// Mitsubishi GX Works2 project: PLC_GROUP12   PLC: FX3G

// global labels: Global1
VAR_GLOBAL
  startDay AT X007 : BOOL;
  WorkingDay AT Y007 : BOOL;
  EmergencySwitch AT X005 : BOOL;
  IceCreamMake AT X001 : BOOL;
END_VAR
VAR_GLOBAL CONSTANT
  Div_Mul_400 : REAL := 400;
END_VAR
VAR_GLOBAL
  regularIceLight AT M10 : BOOL;
END_VAR
VAR_GLOBAL CONSTANT
  MaxForRegular_5 : REAL := 5;
END_VAR
VAR_GLOBAL
  typeInput AT D1300 : REAL;
  analog_Input1 AT D8280 : INT;
  pinukIceLight AT M11 : BOOL;
  PetelAmount AT D1400 : REAL;
  LimonAmount AT D1410 : REAL;
  StableAmount AT D1420 : REAL;
  GummyAmount AT D1430 : REAL;
END_VAR
VAR_GLOBAL CONSTANT
  BearsForRegular_28 : REAL := 28;
END_VAR
VAR_GLOBAL
  EnoughForRegular AT M5 : BOOL;
END_VAR
VAR_GLOBAL CONSTANT
  BearsForPinuk_70 : REAL := 70;
END_VAR
VAR_GLOBAL
  EnoughForPinuk AT M6 : BOOL;
  PetelIcecream AT D1500 : REAL;
END_VAR
VAR_GLOBAL CONSTANT
  PetelIcecream_R_350 : REAL := 350;
  LemonIcecream_R_490 : REAL := 490;
END_VAR
VAR_GLOBAL
  LemonIcecream AT D1510 : REAL;
  StartMakingRegular AT M21 : BOOL;
END_VAR
VAR_GLOBAL CONSTANT
  PetelIcecream_P_560 : REAL := 560;
  LemonIcecream_P_700 : REAL := 700;
  LemonForRegular_455 : REAL := 455;
  StableForRegular_105 : REAL := 105;
END_VAR
VAR_GLOBAL
  subInvRegular AT M7 : BOOL;
  subInvPinuk AT M8 : BOOL;
END_VAR
VAR_GLOBAL CONSTANT
  PetelForPinuk_385 : REAL := 385;
  LemonForPinuk_665 : REAL := 665;
  StableForPinuk_210 : REAL := 210;
  IceCreamTimer_50 : INT := 50;
END_VAR
VAR_GLOBAL
  TimerForIceCream AT TC1 : BOOL;
  FinishedIceCream AT TS1 : BOOL;
  IceCreamMakeLight AT Y000 : BOOL;
  StartMakingPinuk AT M22 : BOOL;
  startFridge AT X002 : BOOL;
  PetelFridge AT D1600 : REAL;
  LemonFridge AT D1610 : REAL;
  MoveToFridge AT M23 : BOOL;
END_VAR
VAR_GLOBAL CONSTANT
  FridgeTimer_80 : INT := 80;
END_VAR
VAR_GLOBAL
  TimerForFridge AT TC2 : BOOL;
  FinishedFridge AT TS2 : BOOL;
  tempSensor AT X003 : BOOL;
  IceCreamFridgeLight AT Y002 : BOOL;
END_VAR
VAR_GLOBAL CONSTANT
  MinForPinuk_6 : REAL := 6;
END_VAR
VAR_GLOBAL
  EnoughInventoryPinuk AT M9 : BOOL;
  EnoughInventoryRegular AT M4 : BOOL;
  mixConatainer AT D1666 : REAL;
  BlendRegular AT M30 : BOOL;
  BlendPinuk AT M31 : BOOL;
  StartBlink AT M32 : BOOL;
END_VAR
VAR_GLOBAL CONSTANT
  SingleBlink_3 : INT := 3;
END_VAR
VAR_GLOBAL
  TimerForOneBlinkY5 AT TC3 : BOOL;
  FinishedOneBlinkY5 AT TS3 : BOOL;
  MixLight1 AT Y005 : BOOL;
  TimerForOneBlinkY6 AT TC4 : BOOL;
  FinishedOneBlinkY6 AT TS4 : BOOL;
  MixLight2 AT Y006 : BOOL;
  FinishedBlendReg AT TS5 : BOOL;
  TimerForBlendReg AT TC5 : BOOL;
END_VAR
VAR_GLOBAL CONSTANT
  BlinkRegular_30 : INT := 30;
END_VAR
VAR_GLOBAL
  BlinkRegular AT M45 : BOOL;
  BlinkPinuk AT M46 : BOOL;
  FinishedBlendPinuk AT TS6 : BOOL;
END_VAR
VAR_GLOBAL CONSTANT
  BlinkPinuk_50 : INT := 50;
END_VAR
VAR_GLOBAL
  TimerForBlendPinuk AT TC6 : BOOL;
  StartPacking AT X004 : BOOL;
  GummyPack AT X000 : BOOL;
  CounterForPacking AT CC1 : BOOL;
END_VAR
VAR_GLOBAL CONSTANT
  UnitsCounter_7 : INT := 7;
END_VAR
VAR_GLOBAL
  FinishedPacking AT CS1 : BOOL;
  PackUnit AT Y004 : BOOL;
  Storage AT D1700 : REAL;
END_VAR
VAR_GLOBAL CONSTANT
  ReadyPackage_1 : REAL := 1;
  OutputDivider_10 : REAL := 10;
END_VAR
VAR_GLOBAL
  output AT D1710 : REAL;
  analogOutput AT D8282 : INT;
END_VAR
VAR_GLOBAL CONSTANT
  RegularUnit_124 : REAL := 124;
  PinukUnit_190 : REAL := 190;
  PetelForRegular_280 : REAL := 280;
END_VAR
VAR_GLOBAL
  EndIteration AT M59 : BOOL;
  NoInventory AT M60 : BOOL;
  RegistorZero AT D1800 : REAL;
  RegZero AT D1810 : INT;
END_VAR
VAR_GLOBAL CONSTANT
  PetelForRegular_279 : REAL := 279;
  LemonForRegular_454 : REAL := 454;
  StableForRegular_104 : REAL := 104;
  BearsForRegular_27 : REAL := 27;
END_VAR

// task Task_01 (event TRUE, interval 0, priority 31): POU_01

PROGRAM POU_01
(* structured ladder/FBD written out as ST: instructions are called as NAME(EN, inputs, outputs); _pN, _eN, _tN stand for wires *)
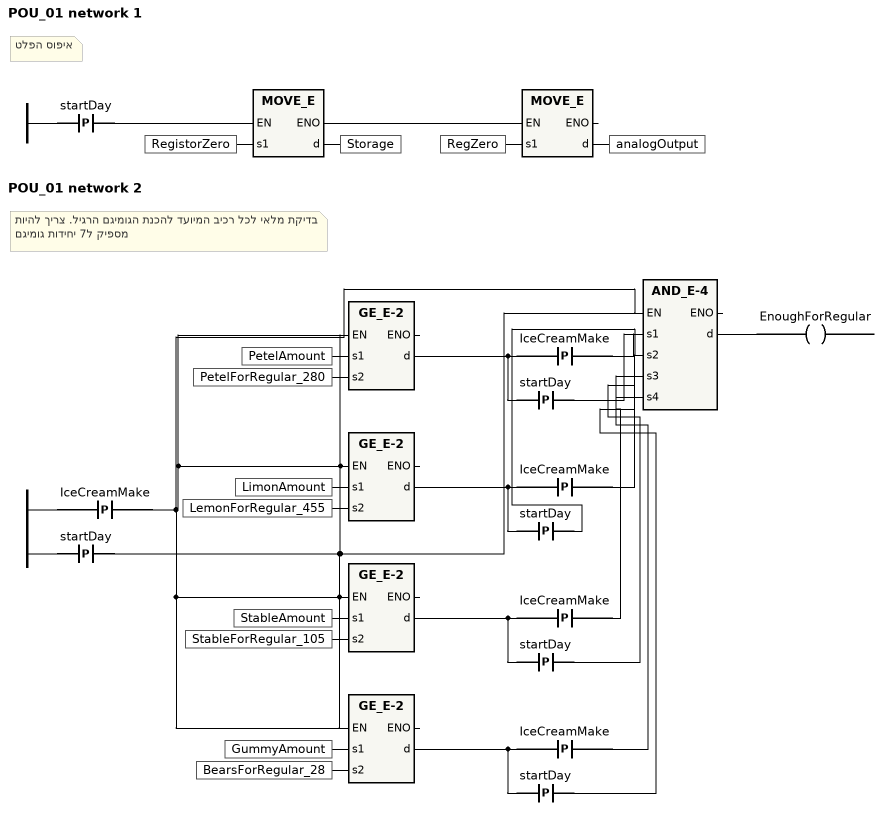
(* network 1 *)
(* איפוס הפלט *)
_e1 := MOVE_E(LDP(TRUE, startDay), RegistorZero, Storage);
MOVE_E(_e1, RegZero, analogOutput);
(* network 2 *)
(* בדיקת מלאי לכל רכיב המיועד להכנת הגומיגם הרגיל. צריך להיות מספיק ל7 יחידות גומיגם *)
_p1 := LDP(TRUE, IceCreamMake) OR LDP(TRUE, startDay);
GE_E(_p1, PetelAmount, PetelForRegular_280, _t2);
GE_E(_p1, LimonAmount, LemonForRegular_455, _t3);
GE_E(_p1, StableAmount, StableForRegular_105, _t4);
GE_E(_p1, GummyAmount, BearsForRegular_28, _t5);
AND_E(_p1, (_t2 AND LDP(TRUE, IceCreamMake)) OR (_t2 AND LDP(TRUE, startDay)), (_t3 AND LDP(TRUE, IceCreamMake)) OR (_t3 AND LDP(TRUE, startDay)), (_t4 AND LDP(TRUE, IceCreamMake)) OR (_t4 AND LDP(TRUE, startDay)), (_t5 AND LDP(TRUE, IceCreamMake)) OR (_t5 AND LDP(TRUE, startDay)), _t6);
EnoughForRegular := _t6;
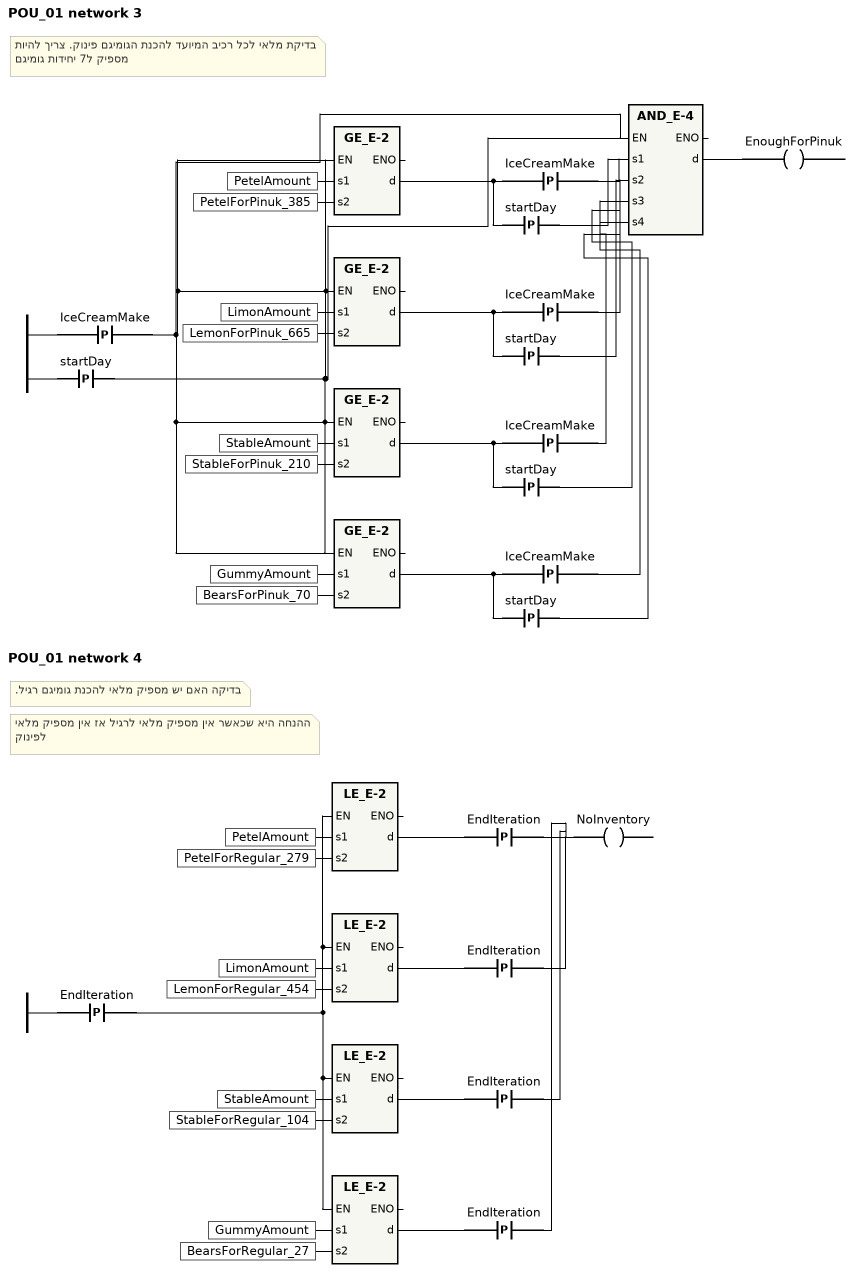
(* network 3 *)
(* בדיקת מלאי לכל רכיב המיועד להכנת הגומיגם פינוק. צריך להיות מספיק ל7 יחידות גומיגם *)
_p1 := LDP(TRUE, IceCreamMake) OR LDP(TRUE, startDay);
GE_E(_p1, PetelAmount, PetelForPinuk_385, _t2);
GE_E(_p1, LimonAmount, LemonForPinuk_665, _t3);
GE_E(_p1, StableAmount, StableForPinuk_210, _t4);
GE_E(_p1, GummyAmount, BearsForPinuk_70, _t5);
AND_E(_p1, (_t2 AND LDP(TRUE, IceCreamMake)) OR (_t2 AND LDP(TRUE, startDay)), (_t3 AND LDP(TRUE, IceCreamMake)) OR (_t3 AND LDP(TRUE, startDay)), (_t4 AND LDP(TRUE, IceCreamMake)) OR (_t4 AND LDP(TRUE, startDay)), (_t5 AND LDP(TRUE, IceCreamMake)) OR (_t5 AND LDP(TRUE, startDay)), _t6);
EnoughForPinuk := _t6;
(* network 4 *)
(* בדיקה האם יש מספיק מלאי להכנת גומיגם רגיל. *)
(* ההנחה היא שכאשר אין מספיק מלאי לרגיל אז אין מספיק מלאי לפינוק *)
_p1 := LDP(TRUE, EndIteration);
LE_E(_p1, PetelAmount, PetelForRegular_279, _t2);
LE_E(_p1, LimonAmount, LemonForRegular_454, _t3);
LE_E(_p1, StableAmount, StableForRegular_104, _t4);
LE_E(_p1, GummyAmount, BearsForRegular_27, _t5);
NoInventory := (_t2 AND LDP(TRUE, EndIteration)) OR (_t3 AND LDP(TRUE, EndIteration)) OR (_t4 AND LDP(TRUE, EndIteration)) OR (_t5 AND LDP(TRUE, EndIteration));
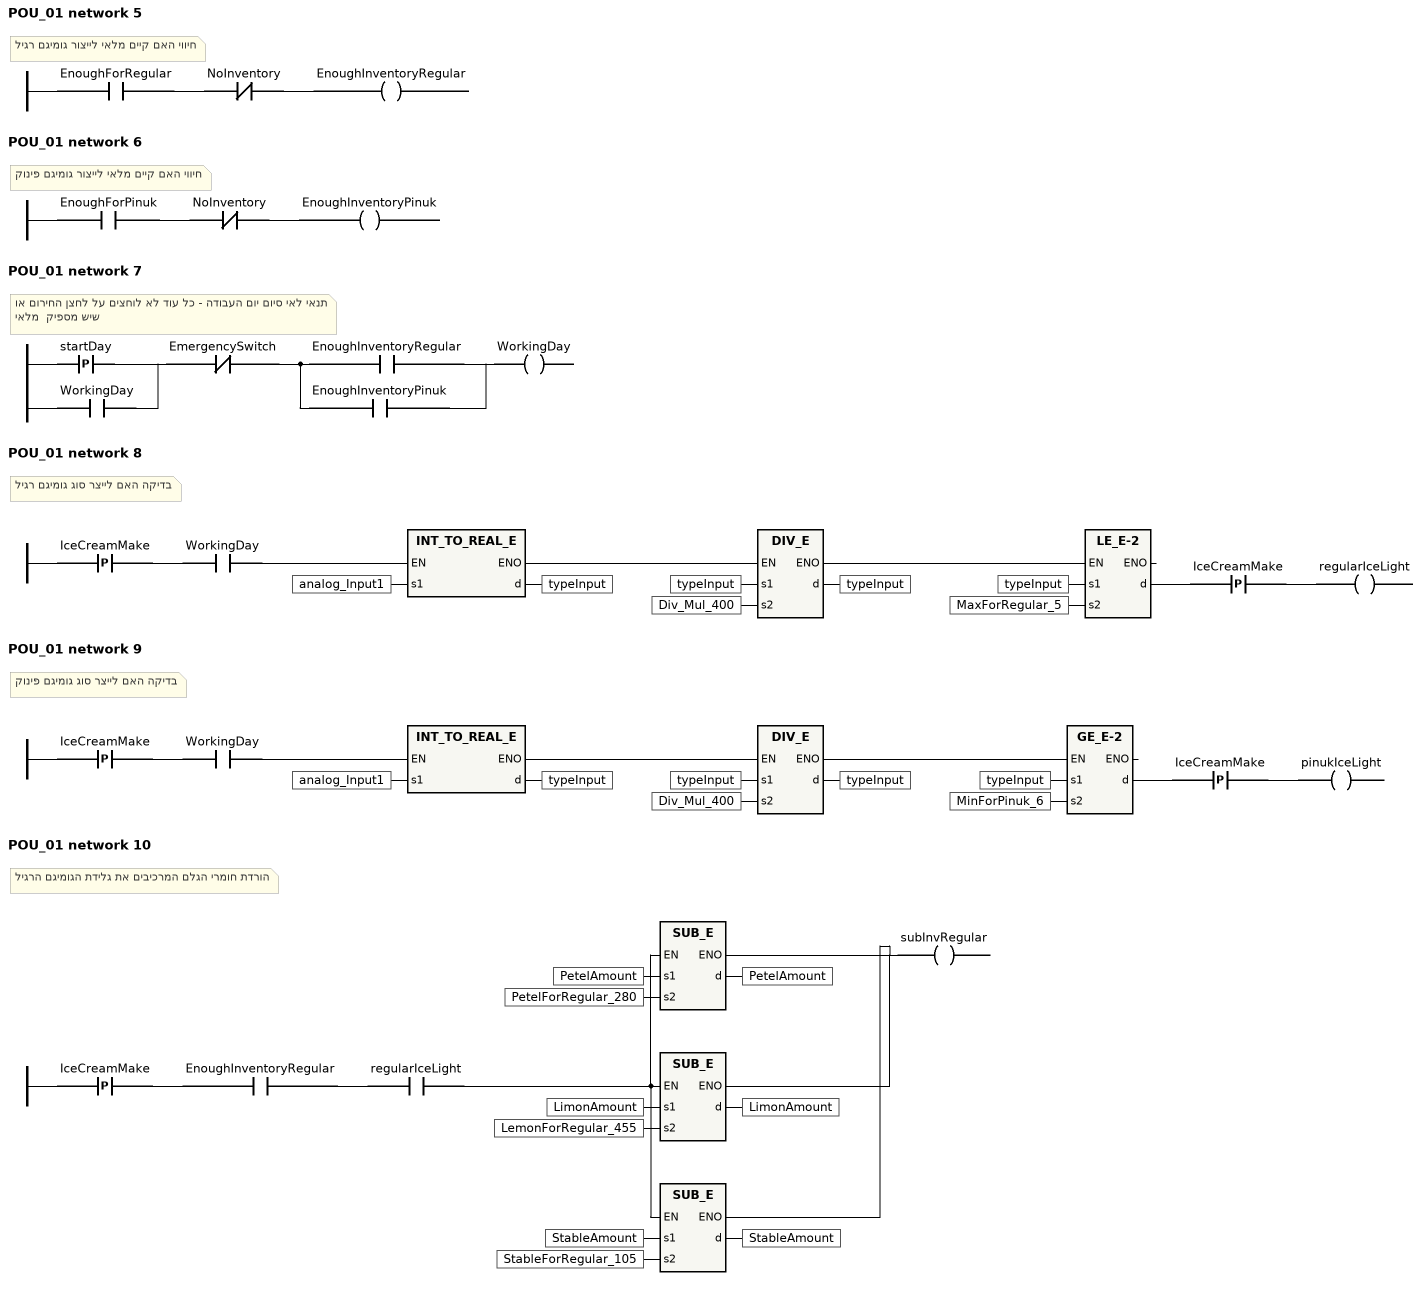
(* network 5 *)
(* חיווי האם קיים מלאי לייצור גומיגם רגיל *)
EnoughInventoryRegular := EnoughForRegular AND NOT NoInventory;
(* network 6 *)
(* חיווי האם קיים מלאי לייצור גומיגם פינוק *)
EnoughInventoryPinuk := EnoughForPinuk AND NOT NoInventory;
(* network 7 *)
(* תנאי לאי סיום יום העבודה - כל עוד לא לוחצים על לחצן החירום או שיש מספיק  מלאי *)
_p1 := (LDP(TRUE, startDay) OR WorkingDay) AND NOT EmergencySwitch;
WorkingDay := (_p1 AND EnoughInventoryRegular) OR (_p1 AND EnoughInventoryPinuk);
(* network 8 *)
(* בדיקה האם לייצר סוג גומיגם רגיל *)
_e1 := INT_TO_REAL_E(LDP(TRUE, IceCreamMake) AND WorkingDay, analog_Input1, typeInput);
_e2 := DIV_E(_e1, typeInput, Div_Mul_400, typeInput);
LE_E(_e2, typeInput, MaxForRegular_5, _t3);
regularIceLight := _t3 AND LDP(TRUE, IceCreamMake);
(* network 9 *)
(* בדיקה האם לייצר סוג גומיגם פינוק *)
_e1 := INT_TO_REAL_E(LDP(TRUE, IceCreamMake) AND WorkingDay, analog_Input1, typeInput);
_e2 := DIV_E(_e1, typeInput, Div_Mul_400, typeInput);
GE_E(_e2, typeInput, MinForPinuk_6, _t3);
pinukIceLight := _t3 AND LDP(TRUE, IceCreamMake);
(* network 10 *)
(* הורדת חומרי הגלם המרכיבים את גלידת הגומיגם הרגיל *)
_p1 := LDP(TRUE, IceCreamMake) AND EnoughInventoryRegular AND regularIceLight;
_e2 := SUB_E(_p1, PetelAmount, PetelForRegular_280, PetelAmount);
_e3 := SUB_E(_p1, LimonAmount, LemonForRegular_455, LimonAmount);
_e4 := SUB_E(_p1, StableAmount, StableForRegular_105, StableAmount);
subInvRegular := _e2 OR _e3 OR _e4;
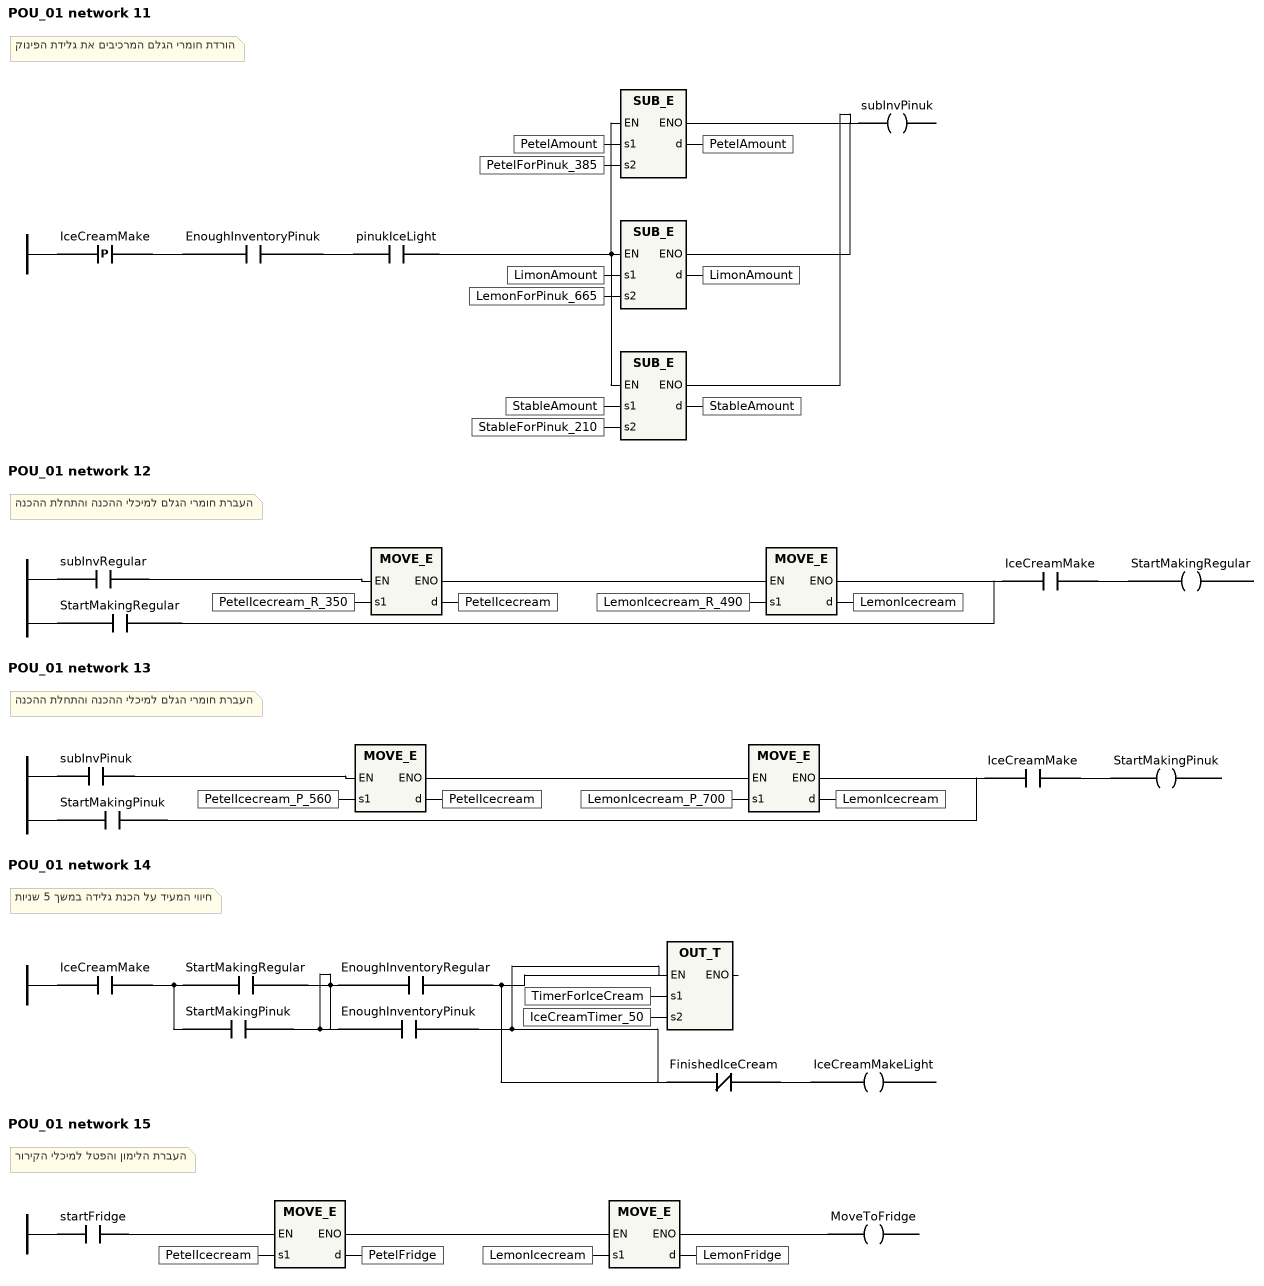
(* network 11 *)
(* הורדת חומרי הגלם המרכיבים את גלידת הפינוק *)
_p1 := LDP(TRUE, IceCreamMake) AND EnoughInventoryPinuk AND pinukIceLight;
_e2 := SUB_E(_p1, PetelAmount, PetelForPinuk_385, PetelAmount);
_e3 := SUB_E(_p1, LimonAmount, LemonForPinuk_665, LimonAmount);
_e4 := SUB_E(_p1, StableAmount, StableForPinuk_210, StableAmount);
subInvPinuk := _e2 OR _e3 OR _e4;
(* network 12 *)
(* העברת חומרי הגלם למיכלי ההכנה והתחלת ההכנה *)
_e1 := MOVE_E(subInvRegular, PetelIcecream_R_350, PetelIcecream);
_e2 := MOVE_E(_e1, LemonIcecream_R_490, LemonIcecream);
StartMakingRegular := (_e2 OR StartMakingRegular) AND IceCreamMake;
(* network 13 *)
(* העברת חומרי הגלם למיכלי ההכנה והתחלת ההכנה *)
_e1 := MOVE_E(subInvPinuk, PetelIcecream_P_560, PetelIcecream);
_e2 := MOVE_E(_e1, LemonIcecream_P_700, LemonIcecream);
StartMakingPinuk := (_e2 OR StartMakingPinuk) AND IceCreamMake;
(* network 14 *)
(* חיווי המעיד על הכנת גלידה במשך 5 שניות *)
_p1 := (IceCreamMake AND StartMakingRegular) OR (IceCreamMake AND StartMakingPinuk);
_p2 := (_p1 AND EnoughInventoryRegular) OR (_p1 AND EnoughInventoryPinuk);
IceCreamMakeLight := _p2 AND NOT FinishedIceCream;
OUT_T(_p2, TimerForIceCream, IceCreamTimer_50);
(* network 15 *)
(* העברת הלימון והפטל למיכלי הקירור *)
_e1 := MOVE_E(startFridge, PetelIcecream, PetelFridge);
_e2 := MOVE_E(_e1, LemonIcecream, LemonFridge);
MoveToFridge := _e2;
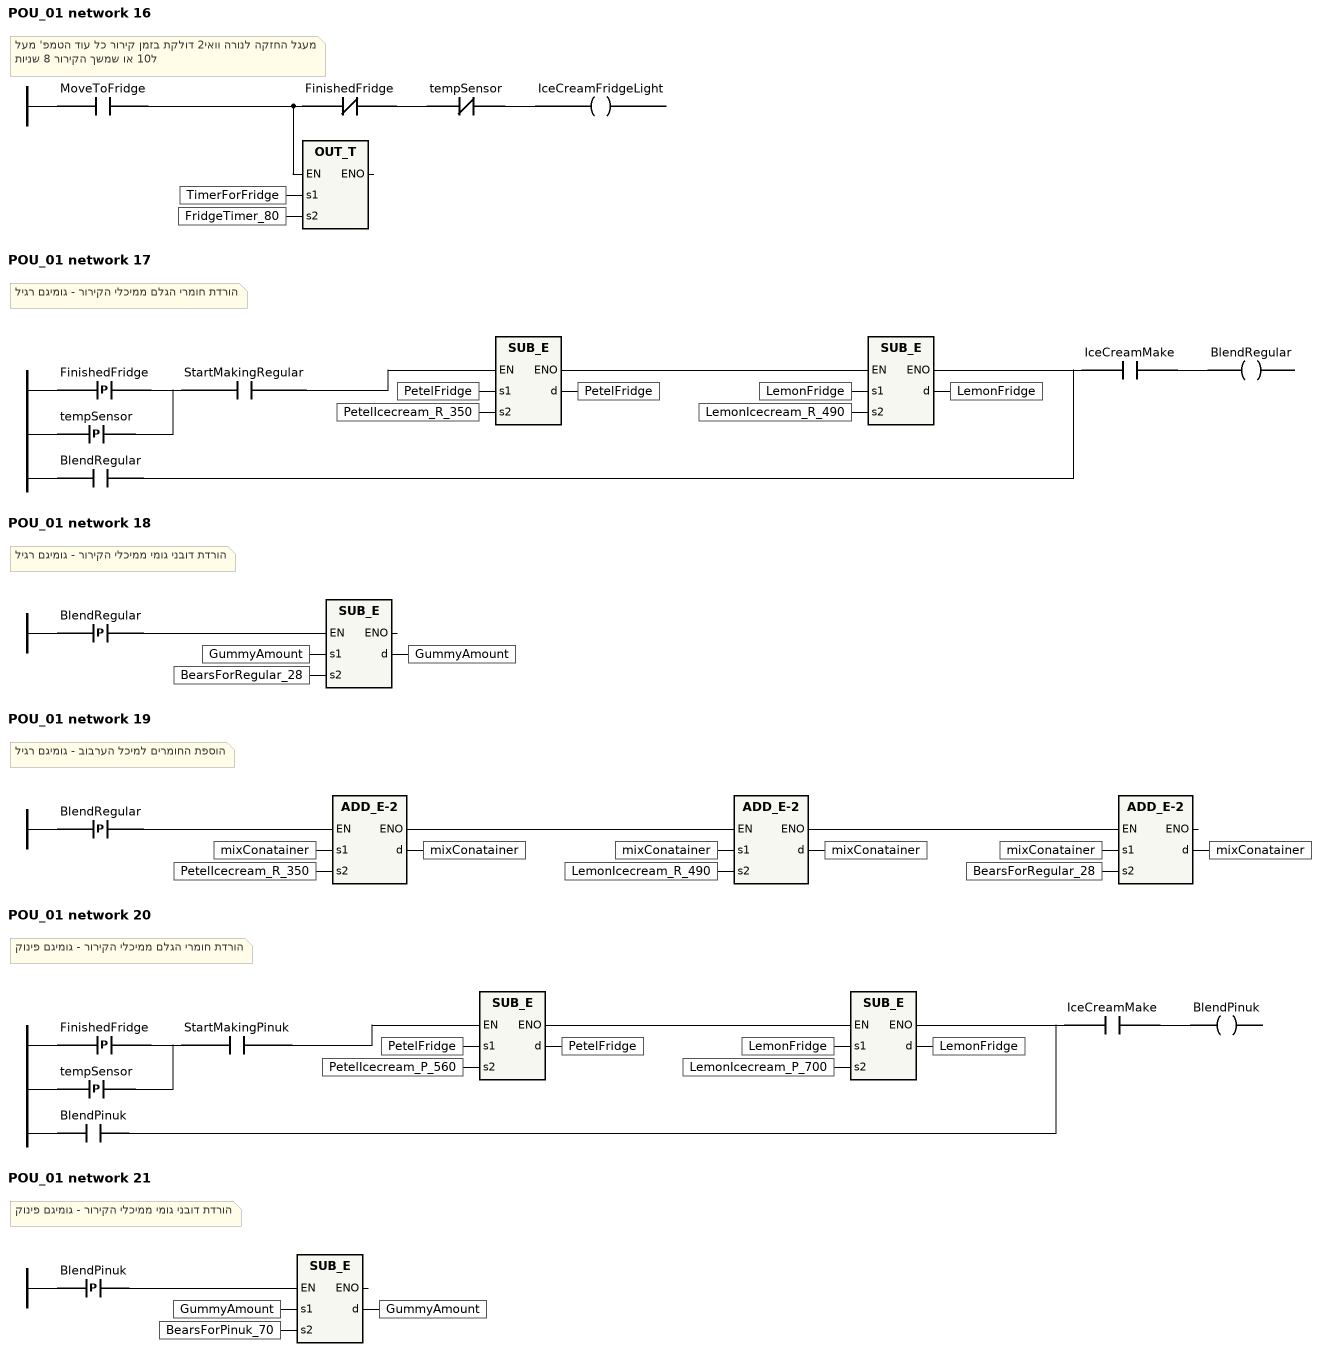
(* network 16 *)
(* מעגל החזקה לנורה וואי2 דולקת בזמן קירור כל עוד הטמפ' מעל ל10 או שמשך הקירור 8 שניות *)
IceCreamFridgeLight := MoveToFridge AND NOT FinishedFridge AND NOT tempSensor;
OUT_T(MoveToFridge, TimerForFridge, FridgeTimer_80);
(* network 17 *)
(* הורדת חומרי הגלם ממיכלי הקירור - גומיגם רגיל *)
_e1 := SUB_E((LDP(TRUE, FinishedFridge) OR LDP(TRUE, tempSensor)) AND StartMakingRegular, PetelFridge, PetelIcecream_R_350, PetelFridge);
_e2 := SUB_E(_e1, LemonFridge, LemonIcecream_R_490, LemonFridge);
BlendRegular := (_e2 OR BlendRegular) AND IceCreamMake;
(* network 18 *)
(* הורדת דובני גומי ממיכלי הקירור - גומיגם רגיל *)
SUB_E(LDP(TRUE, BlendRegular), GummyAmount, BearsForRegular_28, GummyAmount);
(* network 19 *)
(* הוספת החומרים למיכל הערבוב - גומיגם רגיל *)
_e1 := ADD_E(LDP(TRUE, BlendRegular), mixConatainer, PetelIcecream_R_350, mixConatainer);
_e2 := ADD_E(_e1, mixConatainer, LemonIcecream_R_490, mixConatainer);
ADD_E(_e2, mixConatainer, BearsForRegular_28, mixConatainer);
(* network 20 *)
(* הורדת חומרי הגלם ממיכלי הקירור - גומיגם פינוק *)
_e1 := SUB_E((LDP(TRUE, FinishedFridge) OR LDP(TRUE, tempSensor)) AND StartMakingPinuk, PetelFridge, PetelIcecream_P_560, PetelFridge);
_e2 := SUB_E(_e1, LemonFridge, LemonIcecream_P_700, LemonFridge);
BlendPinuk := (_e2 OR BlendPinuk) AND IceCreamMake;
(* network 21 *)
(* הורדת דובני גומי ממיכלי הקירור - גומיגם פינוק *)
SUB_E(LDP(TRUE, BlendPinuk), GummyAmount, BearsForPinuk_70, GummyAmount);
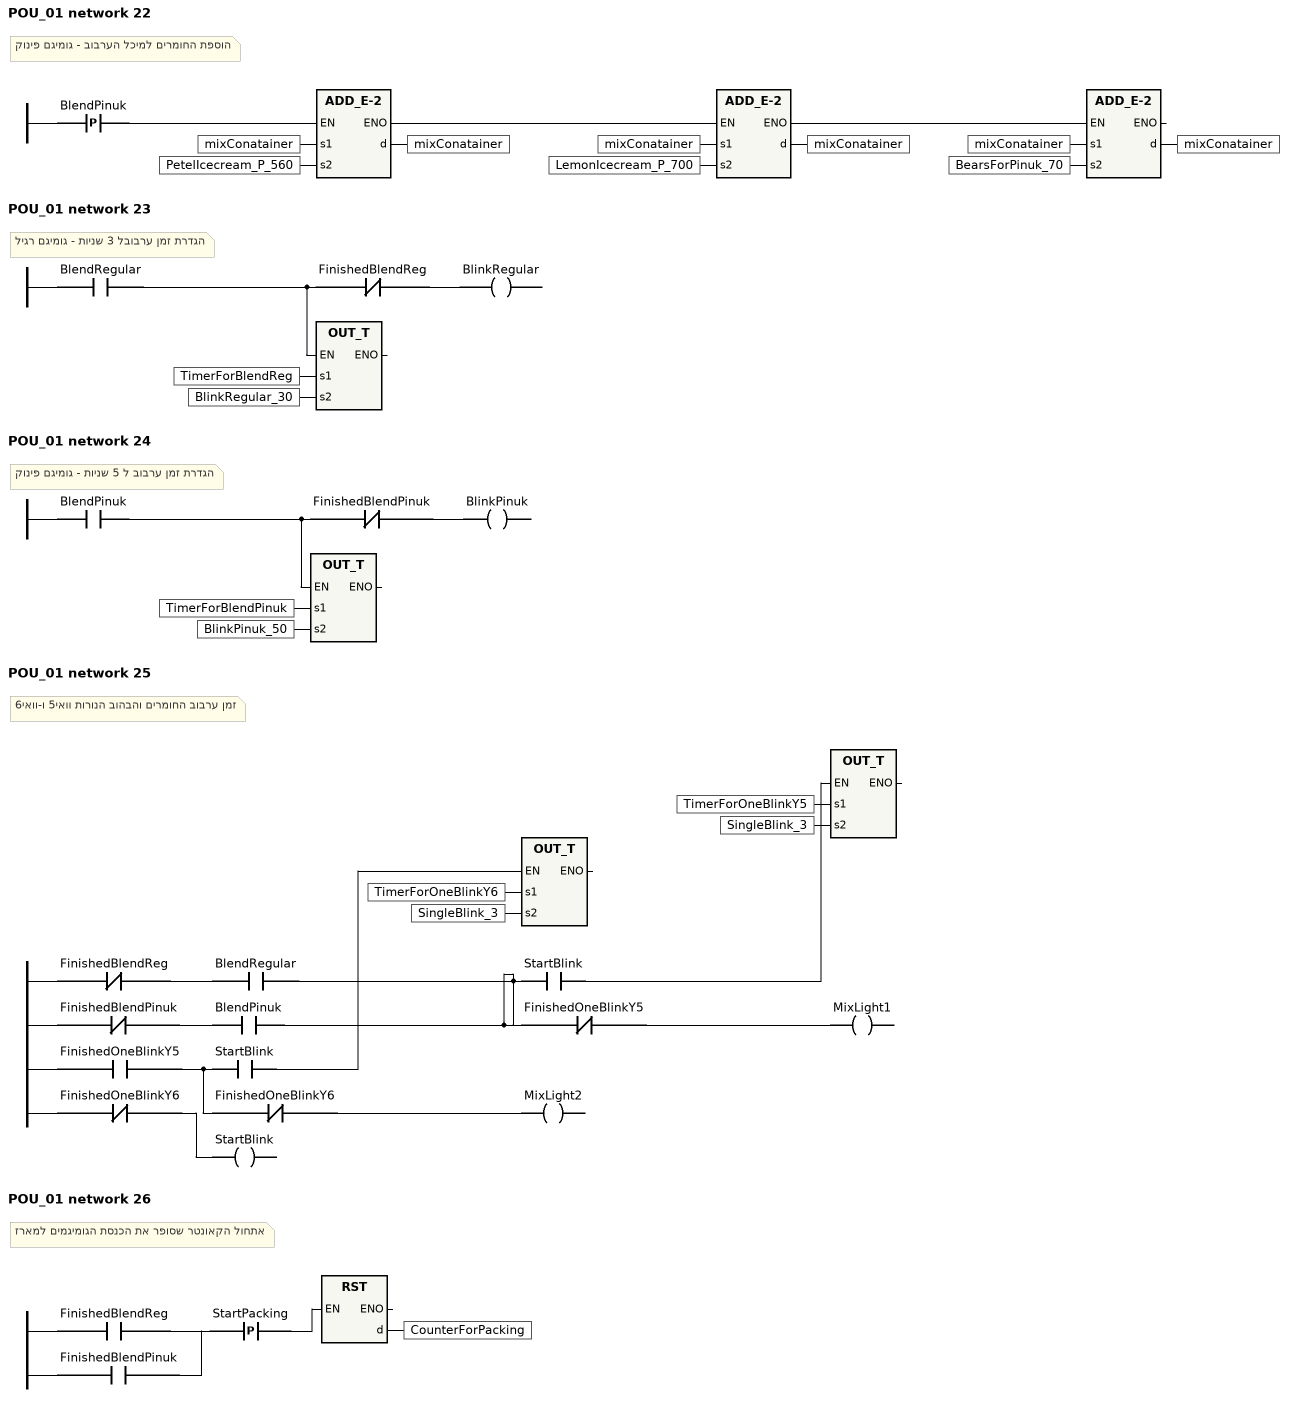
(* network 22 *)
(* הוספת החומרים למיכל הערבוב - גומיגם פינוק *)
_e1 := ADD_E(LDP(TRUE, BlendPinuk), mixConatainer, PetelIcecream_P_560, mixConatainer);
_e2 := ADD_E(_e1, mixConatainer, LemonIcecream_P_700, mixConatainer);
ADD_E(_e2, mixConatainer, BearsForPinuk_70, mixConatainer);
(* network 23 *)
(* הגדרת זמן ערבובל 3 שניות - גומיגם רגיל *)
BlinkRegular := BlendRegular AND NOT FinishedBlendReg;
OUT_T(BlendRegular, TimerForBlendReg, BlinkRegular_30);
(* network 24 *)
(* הגדרת זמן ערבוב ל 5 שניות - גומיגם פינוק *)
BlinkPinuk := BlendPinuk AND NOT FinishedBlendPinuk;
OUT_T(BlendPinuk, TimerForBlendPinuk, BlinkPinuk_50);
(* network 25 *)
(* זמן ערבוב החומרים והבהוב הנורות וואי5 ו-וואי6 *)
_p1 := (NOT FinishedBlendReg AND BlendRegular) OR (NOT FinishedBlendPinuk AND BlendPinuk);
OUT_T(_p1 AND StartBlink, TimerForOneBlinkY5, SingleBlink_3);
MixLight1 := _p1 AND NOT FinishedOneBlinkY5;
OUT_T(FinishedOneBlinkY5 AND StartBlink, TimerForOneBlinkY6, SingleBlink_3);
MixLight2 := FinishedOneBlinkY5 AND NOT FinishedOneBlinkY6;
StartBlink := NOT FinishedOneBlinkY6;
(* network 26 *)
(* אתחול הקאונטר שסופר את הכנסת הגומיגמים למארז *)
RST((FinishedBlendReg OR FinishedBlendPinuk) AND LDP(TRUE, StartPacking), CounterForPacking);
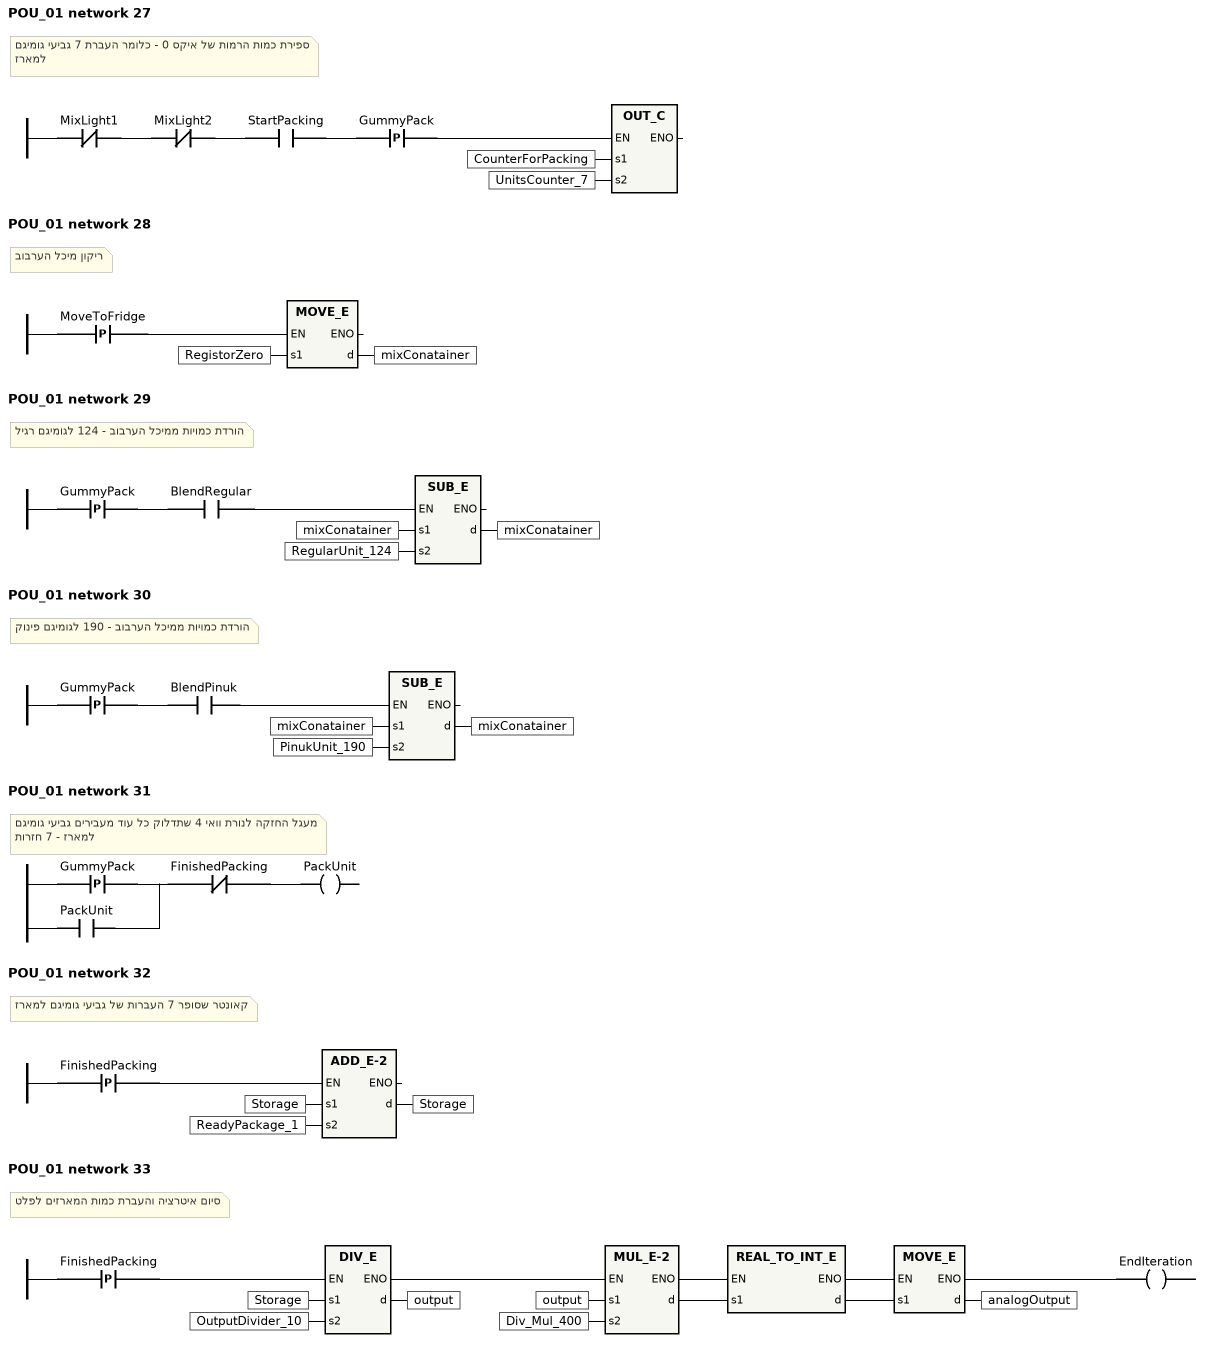
(* network 27 *)
(* ספירת כמות הרמות של איקס 0 - כלומר העברת 7 גביעי גומיגם למארז *)
OUT_C(NOT MixLight1 AND NOT MixLight2 AND StartPacking AND LDP(TRUE, GummyPack), CounterForPacking, UnitsCounter_7);
(* network 28 *)
(* ריקון מיכל הערבוב *)
MOVE_E(LDP(TRUE, MoveToFridge), RegistorZero, mixConatainer);
(* network 29 *)
(* הורדת כמויות ממיכל הערבוב - 124 לגומיגם רגיל *)
SUB_E(LDP(TRUE, GummyPack) AND BlendRegular, mixConatainer, RegularUnit_124, mixConatainer);
(* network 30 *)
(* הורדת כמויות ממיכל הערבוב - 190 לגומיגם פינוק *)
SUB_E(LDP(TRUE, GummyPack) AND BlendPinuk, mixConatainer, PinukUnit_190, mixConatainer);
(* network 31 *)
(* מעגל החזקה לנורת וואי 4 שתדלוק כל עוד מעבירים גביעי גומיגם למארז - 7 חזרות *)
PackUnit := (LDP(TRUE, GummyPack) OR PackUnit) AND NOT FinishedPacking;
(* network 32 *)
(* קאונטר שסופר 7 העברות של גביעי גומיגם למארז *)
ADD_E(LDP(TRUE, FinishedPacking), Storage, ReadyPackage_1, Storage);
(* network 33 *)
(* סיום איטרציה והעברת כמות המארזים לפלט *)
_e1 := DIV_E(LDP(TRUE, FinishedPacking), Storage, OutputDivider_10, output);
_e3 := MUL_E(_e1, output, Div_Mul_400, _t2);
_e5 := REAL_TO_INT_E(_e3, _t2, _t4);
_e6 := MOVE_E(_e5, _t4, analogOutput);
EndIteration := _e6;
END_PROGRAM
